{attribute 'no_explicit_call' := 'do not call this FB directly'}{attribute 'enable_dynamic_creation'}
FUNCTION_BLOCK FINAL Node_Literal_Generic EXTENDS Node
VAR
	value : I_Datatype;
	out : I_Datatype;
END_VAR

METHOD PUBLIC Clone : I_Node
VAR
	pointerToNode : POINTER TO Node_Literal_BOOL;
END_VAR
pointerToNode := __NEW(Node_Literal_BOOL);
Clone := pointerToNode^;
END_METHOD

METHOD ConfigureDatatype
VAR_INPUT
	Datatype : I_Datatype;
END_VAR
value := Datatype.clone();
out := Datatype.clone();


IF NOT Datatype.TryResolveStructure(myStructure) THEN
	RETURN;
END_IF

myStructure.
END_METHOD

METHOD PROTECTED OnExecute : HRESULT
VAR
END_VAR
out.TryCopyFrom(value);
END_METHOD

END_FUNCTION_BLOCK

(* stored: Version 1.1.0.1, ProductVersion 3.1.4024.12
   POU Node_Literal_Generic: Id {693e78a4-fc28-4994-a2ff-3e9a5cf1df5b}, SpecialFunc None
   Method Clone: Id {0f740e25-6053-4b99-8d9b-fa967d06c198}
   Method ConfigureDatatype: Id {77fbf8b0-331d-4185-8a53-db5bff7ebe75}
   Method OnExecute: Id {c9463d74-43af-44d9-83d8-f8b33f77ad74} *)
